Fanuc KAREL source: MP0094.KL

PROGRAM MP0094
%STACKSIZE=65535
%PRIORITY=65535
%NOLOCKGROUP
ROUTINE FINT(P1 : INTEGER) : INTEGER FROM MP0094
ROUTINE FREAL(P1 : REAL) : REAL FROM MP0094
ROUTINE RTEST(P1 : INTEGER; P2 : REAL) FROM MP0094
ROUTINE FINT
BEGIN
RETURN((P1 + 1))
END FINT
ROUTINE FREAL
BEGIN
RETURN((P1 + 1.0))
END FREAL
ROUTINE RTEST
VAR
U2C_1 : INTEGER
U2C_2 : INTEGER
U2C_3 : INTEGER
S1 : REAL
U2C_5 : INTEGER
U2C_6 : REAL
U2C_7 : REAL
S2 : REAL
BEGIN
U2C_1=7
U2C_2=3
U2C_3=2
S1=2.5
U2C_5=1083179008
U2C_6=1.5
-- UNSAFE_SOURCE_IR line 28: CALL_RESULT FREAL(S1)
END RTEST
BEGIN
RTEST(7,2.5)
END MP0094
